FUNCTION AGILOG_DebugStop : BOOL

GVL_RunTimeLogger.g_debugLogFileName  := 'defaultLogFileName.txt';

GVL_RunTimeLogger.g_enableDebugLog := FALSE;

END_FUNCTION

(* stored: Version 1.1.0.1, ProductVersion 3.1.4024.12
   POU AGILOG_DebugStop: Id {ba7aeb2d-6599-472f-838a-f2d60329c612}, SpecialFunc None *)
